FUNCTION_BLOCK AX_SPLIT_3 (* SPLIT 1 AX into 3 AX *)
  (* Standard: 61499-2; Description: Copyright (c) 2025 HR Agrartechnik GmbH This program and the accompanying materials are made available under the terms of the Eclipse Public License 2.0 which is available at https://www.eclipse.org/legal/epl-2.0/ SPDX-License-Identifier: EPL-2.0 *)
  (* Version 1.0, 2025-01-24, Franz Höpfinger, HR Agrartechnik GmbH *)
  {SET_ATTRIBUTE(eclipse4diac::core::GenericClassName, 'GEN_AX_SPLIT')}
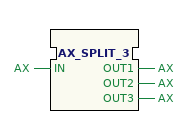
  SOCKETS
    IN : AX;
  END_SOCKETS
  PLUGS
    OUT1 : AX;
    OUT2 : AX;
    OUT3 : AX;
  END_PLUGS
END_FUNCTION_BLOCK
